{attribute 'qualified_only'}
{attribute 'strict'}
TYPE eLightMode :
(
	Init,
	Run,
	Shutdown,
	Error
	
);
END_TYPE

(* stored: Version 1.1.0.1, ProductVersion 3.1.4024.12
   DUT eLightMode: Id {d116aa5f-91b8-497d-b6b0-320babf754aa} *)
